(* Logix 5000 project; controller RG_Chopper vendor 1 type 14 code 235 rev 32.12; software revision 32.04 *)

TASK FLASH_1_SEC (periodic, rate 1000 ms, priority 10, watchdog 1000 ms) : FLASH
TASK MainTask (continuous, watchdog 500 ms) : MainProgram
TASK SafetyTask (periodic, rate 20 ms, priority 5, watchdog 20 ms) : SafetyProgram

MODULES
   Local : vendor 1 type 14 code 235 (5069 0, rev 32.12)
      DBX102_VFD : PowerFlex 525-EENET (Ethernet 10.0.7.41, rev 5.2, Output RPI 20 ms)   // Product Discharge Pump
      DBX104_VFD : PowerFlex 525-EENET (Ethernet 10.0.7.42, rev 5.2, Output RPI 20 ms)   // VFD DBX - 104 - Elevator Drive
           DBX104_VFD:O.Stop   // DBX-104 Drum Dumper VFD Stop
           DBX104_VFD:O.Reverse   // DBX-104 Drum Dumper VFD Direction UP
           DBX104_VFD:O.ClearFaults   // DBX-104 Drum Dumper VFD Clear Faults
           DBX104_VFD:O.Start   // DBX-104 Drum Dumper VFD Start
           DBX104_VFD:O   // DBX-104 Drum Dumper VFD Direction DOWN
      DO_4 : 5069-OB16 (5069 2, rev 2.1, StandardDataDriven RPI 5 ms)   // Digital Output - Slot 4 - 16 point
           Local:2:O.Pt15.Data   // CIP Caustic Request CIP CAUSTIC CR-202
           Local:2:O.Pt14.Data   // CIP Request System Ready CIP Enable CR-201
      DI_S_3 : 5069-IB8S (5069 4, rev 1.1, SafetyInput RPI 20 ms)   // Digital Input Safety - Slot 3 - 8 point
      DI_S_4 : 5069-IB8S (5069 7, rev 1.1, SafetyInput RPI 20 ms)   // Digital Input Safety - Slot 7 - 8 point
      DI_1 : 5069-IB16 (5069 1, rev 2.1, StandardDataDriven RPI 5 ms)   // Digital Input Slot 1 - 16 point
      IO_Link_1 : vendor 322 type 12 code 1123 (Ethernet 10.0.7.71, rev 1.1, StandardDataDriven RPI 10 ms)   // I/O-Link #1 - AL1123
           IO_Link_1:I.Data[207].8   // Port 0 LS-U1
           IO_Link_1:I.Data[207].0   // Port 1 LSS-U2
           IO_Link_1:I.Data[207].10   // Port 4 LS-OT
           IO_Link_1:I.Data[207].1   // Port 3 LS-L1
           IO_Link_1:I.Data[207].9   // Port 2 LSS-L2
      DI_S_2 : 5069-IB8S (5069 3, rev 1.1, SafetyInput RPI 20 ms)   // Digital Input Safety - Slot 2 - 8 point
      DO_S_5 : 5069-OBV8S (5069 5, rev 1.11, SafetyOutput RPI 20 ms, SafetyInput RPI 20 ms)   // Digital Output Safety - Slot 5 - 8 point
           Local:5:O.Pt05.Data   // M104 Elevator Motor Start FORWARD UP (Safety)
           Local:5:O.Pt02.Data   // Reset Button Light
           Local:5:O.Pt03.Data   // Interface Relay Output
           Local:5:O.Pt06.Data   // M104 Elevator Motor Start REVERSE (Safety)
           Local:5:O.Pt04.Data   // M104 Elevator Motor Start (EN) (Safety)
      AO_6 : vendor 1 type 115 code 313 (5069 6, rev 2.1, StandardDataDriven RPI 80 ms)   // Analog Output - Slot 6 - 8 point
END_MODULES

ADD_ON_INSTRUCTION ANLG_SCALE   (* revision 1.0, vendor JBT Food Tech *)
// Scales an Analog Value
// Revision note:
// Rev 1.0 - 9/9/2010 - KM
VAR_INPUT
   Anlg_In : REAL; {required}
   RAW_Min : REAL; {visible}
   RAW_Max : REAL; {visible}
   EU_Min : REAL; {visible}
   EU_Max : REAL; {visible}
END_VAR
VAR_OUTPUT
   Anlg_Scaled : REAL; {access Read Only, required}
END_VAR

ROUTINE Logic   (* ladder *)
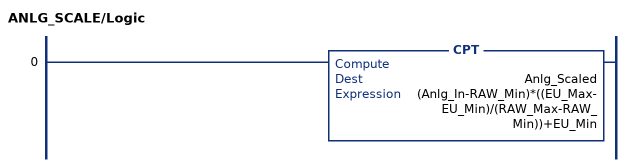
   0: CPT(Anlg_Scaled,(Anlg_In-RAW_Min)*((EU_Max-EU_Min)/(RAW_Max-RAW_Min))+EU_Min);
END_ROUTINE
END_ADD_ON_INSTRUCTION

ADD_ON_INSTRUCTION Generic_4PORT_IOL   (* revision 1.0 *)
// Revision note:
// 4/27/17
VAR_OUTPUT
   Datastorage_Error : BOOL; {access Read Only, visible}
   Device_Not_Connected : BOOL; {access Read Only, visible}
   Invalid_Data : BOOL; {access Read Only, visible}
   IOL_Mode : BOOL; {access Read Only, visible}
END_VAR
VAR_IN_OUT
   PLC_Input : INT[123]; {required}
   PLC_Output : INT[87]; {required}
END_VAR
VAR_INPUT
   Port_Process_Data_Size : INT; {visible}
   Port_Number : INT; {visible}
END_VAR
VAR_OUTPUT
   Process_Data : INT; {access Read Only}
   Wrong_VID_DID : BOOL; {access Read Only, visible}
   IN_Data1 : INT; {visible}
   IN_Data2 : INT; {visible}
   IN_Data3 : INT; {visible}
   IN_Data4 : INT; {visible}
   Out_Data1 : INT; {visible}
   Out_Data2 : INT; {visible}
   Out_Data3 : INT; {visible}
   Out_Data4 : INT; {visible}
   Vendor_ID : INT; {access Read Only, visible}
   Device_ID : INT; {access Read Only, visible}
END_VAR
VAR
   Data_Size : INT; {access None}
   Offset_Address : INT; {access None}
   Offset_StatusFlgs : INT; {access None}
   Process_Offset : INT; {access None}
   Process_PDI : INT; {access None}
   RealPort_Num : INT; {access None}
   StatusFlgs_Offset : INT; {access None}
   Process_Out_Offset : INT; {access None}
END_VAR

ROUTINE Logic   (* ladder *)
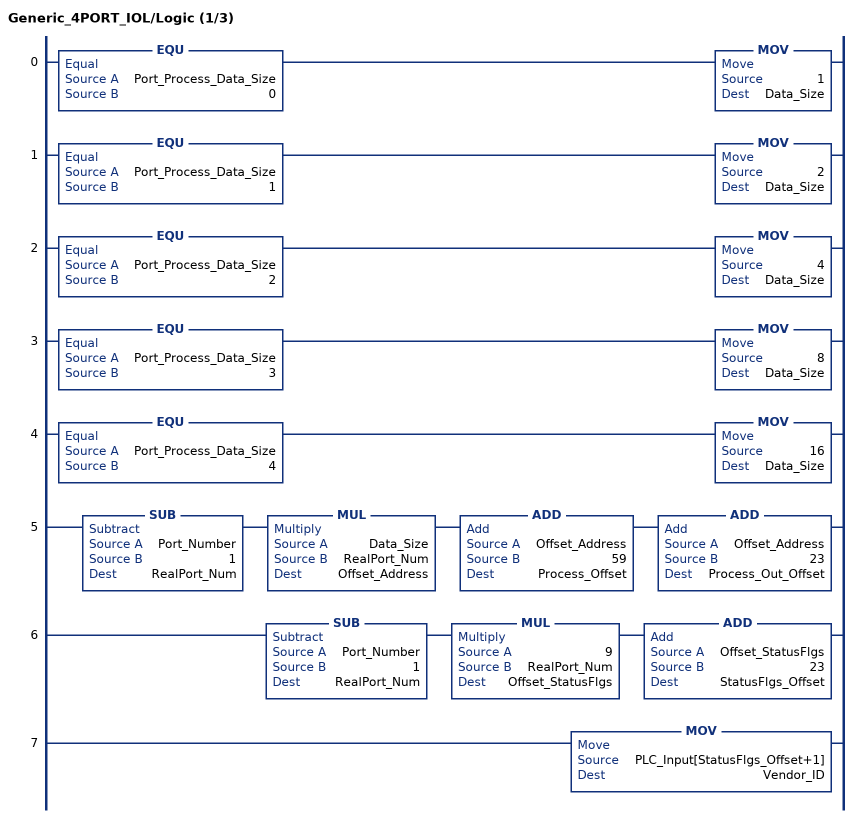
   0: EQU(Port_Process_Data_Size,0)MOV(1,Data_Size);
   1: EQU(Port_Process_Data_Size,1)MOV(2,Data_Size);
   2: EQU(Port_Process_Data_Size,2)MOV(4,Data_Size);
   3: EQU(Port_Process_Data_Size,3)MOV(8,Data_Size);
   4: EQU(Port_Process_Data_Size,4)MOV(16,Data_Size);
   5: SUB(Port_Number,1,RealPort_Num)MUL(Data_Size,RealPort_Num,Offset_Address)ADD(Offset_Address,59,Process_Offset)ADD(Offset_Address,23,Process_Out_Offset);
   6: SUB(Port_Number,1,RealPort_Num)MUL(9,RealPort_Num,Offset_StatusFlgs)ADD(Offset_StatusFlgs,23,StatusFlgs_Offset);
   7: MOV(PLC_Input[StatusFlgs_Offset+1],Vendor_ID);
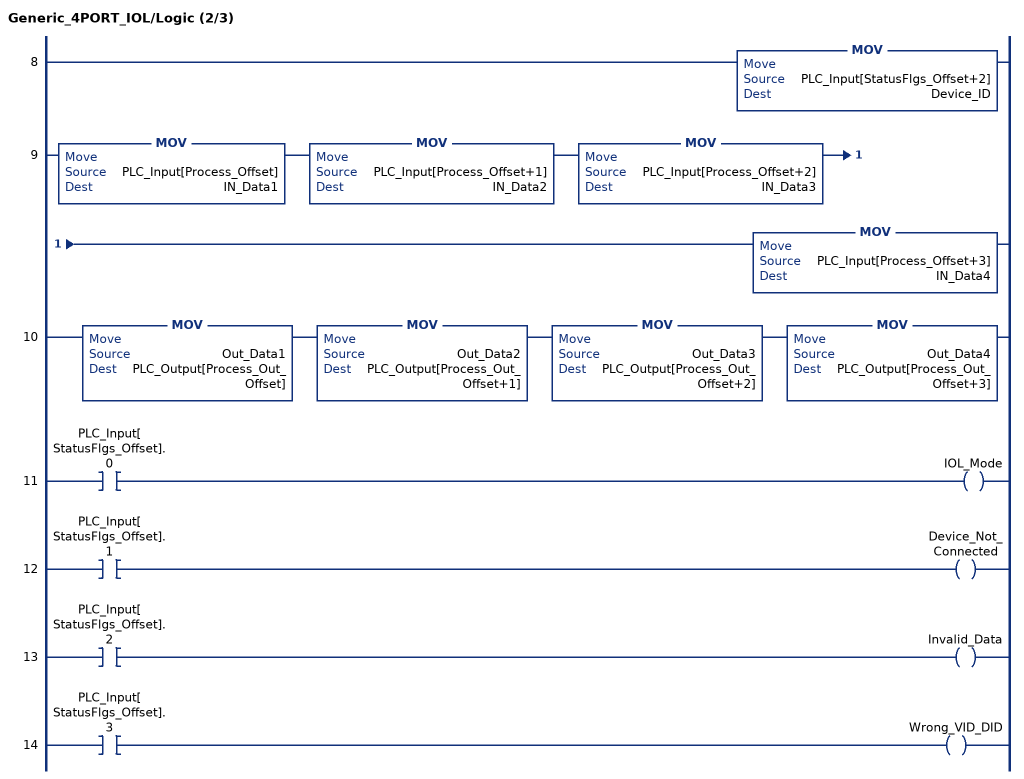
   8: MOV(PLC_Input[StatusFlgs_Offset+2],Device_ID);
   9: MOV(PLC_Input[Process_Offset],IN_Data1)MOV(PLC_Input[Process_Offset+1],IN_Data2)MOV(PLC_Input[Process_Offset+2],IN_Data3)MOV(PLC_Input[Process_Offset+3],IN_Data4);
   10: MOV(Out_Data1,PLC_Output[Process_Out_Offset])MOV(Out_Data2,PLC_Output[Process_Out_Offset+1])MOV(Out_Data3,PLC_Output[Process_Out_Offset+2])MOV(Out_Data4,PLC_Output[Process_Out_Offset+3]);
   11: XIC(PLC_Input[StatusFlgs_Offset].0)OTE(IOL_Mode);
   12: XIC(PLC_Input[StatusFlgs_Offset].1)OTE(Device_Not_Connected);
   13: XIC(PLC_Input[StatusFlgs_Offset].2)OTE(Invalid_Data);
   14: XIC(PLC_Input[StatusFlgs_Offset].3)OTE(Wrong_VID_DID);
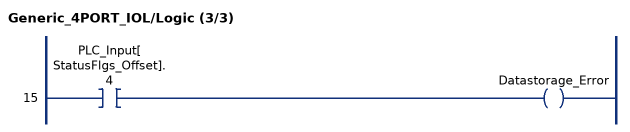
   15: XIC(PLC_Input[StatusFlgs_Offset].4)OTE(Datastorage_Error);
END_ROUTINE
END_ADD_ON_INSTRUCTION

ADD_ON_INSTRUCTION Generic_8PORT_IOL   (* revision 1.0 *)
// Revision note:
// 4/27/17
VAR_OUTPUT
   Datastorage_Error : BOOL; {access Read Only, visible}
   Device_Not_Connected : BOOL; {access Read Only, visible}
   Invalid_Data : BOOL; {access Read Only, visible}
   IOL_Mode : BOOL; {access Read Only, visible}
END_VAR
VAR_IN_OUT
   PLC_Input : INT[223]; {required}
   PLC_Output : INT[151]; {required}
END_VAR
VAR_INPUT
   Port_Process_Data_Size : INT; {visible}
   Port_Number : INT; {visible}
END_VAR
VAR_OUTPUT
   Process_Data : INT; {access Read Only}
   Wrong_VID_DID : BOOL; {access Read Only, visible}
   IN_Data1 : INT; {visible}
   IN_Data2 : INT; {visible}
   IN_Data3 : INT; {visible}
   IN_Data4 : INT; {visible}
   Out_Data1 : INT; {visible}
   Out_Data2 : INT; {visible}
   Out_Data3 : INT; {visible}
   Out_Data4 : INT; {visible}
   Vendor_ID : INT; {access Read Only, visible}
   Device_ID : INT; {access Read Only, visible}
END_VAR
VAR
   Data_Size : INT; {access None}
   Offset_Address : INT; {access None}
   Offset_StatusFlgs : INT; {access None}
   Process_Offset : INT; {access None}
   Process_PDI : INT; {access None}
   RealPort_Num : INT; {access None}
   StatusFlgs_Offset : INT; {access None}
   Process_Out_Offset : INT; {access None}
END_VAR

ROUTINE Logic   (* ladder *)
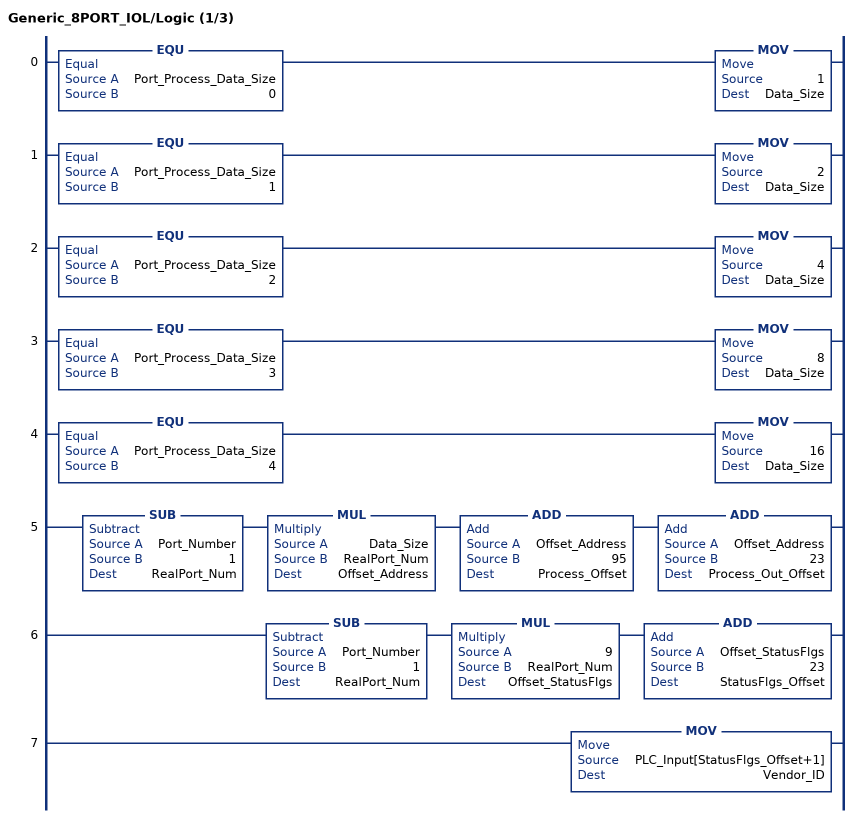
   0: EQU(Port_Process_Data_Size,0)MOV(1,Data_Size);
   1: EQU(Port_Process_Data_Size,1)MOV(2,Data_Size);
   2: EQU(Port_Process_Data_Size,2)MOV(4,Data_Size);
   3: EQU(Port_Process_Data_Size,3)MOV(8,Data_Size);
   4: EQU(Port_Process_Data_Size,4)MOV(16,Data_Size);
   5: SUB(Port_Number,1,RealPort_Num)MUL(Data_Size,RealPort_Num,Offset_Address)ADD(Offset_Address,95,Process_Offset)ADD(Offset_Address,23,Process_Out_Offset);
   6: SUB(Port_Number,1,RealPort_Num)MUL(9,RealPort_Num,Offset_StatusFlgs)ADD(Offset_StatusFlgs,23,StatusFlgs_Offset);
   7: MOV(PLC_Input[StatusFlgs_Offset+1],Vendor_ID);
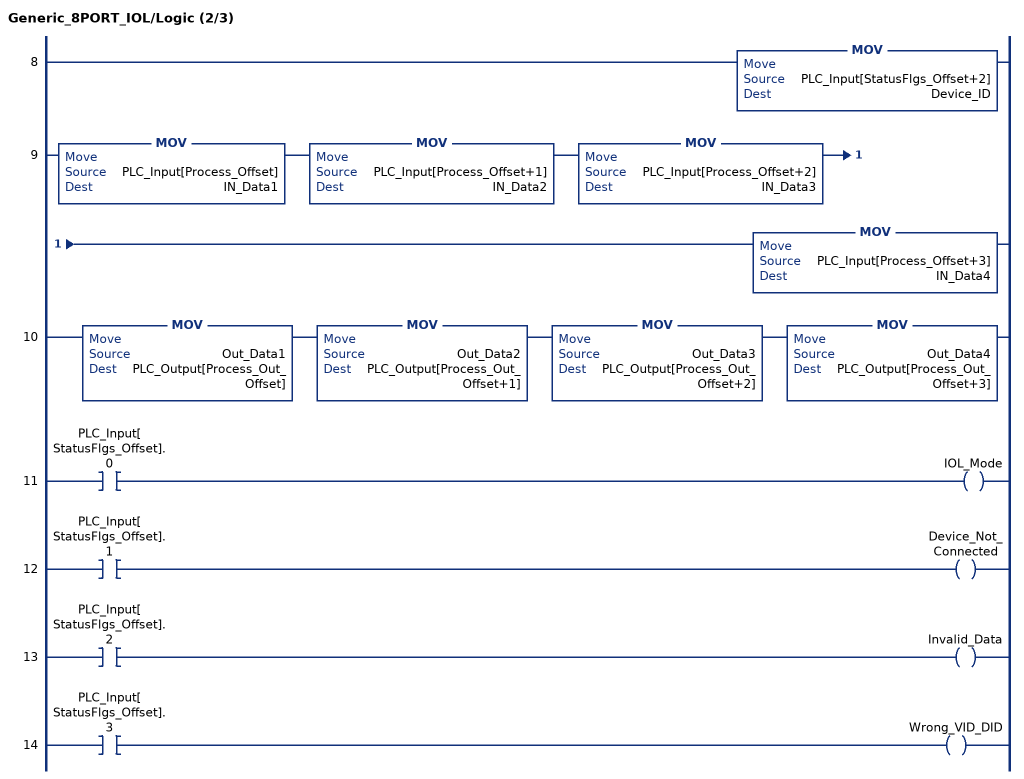
   8: MOV(PLC_Input[StatusFlgs_Offset+2],Device_ID);
   9: MOV(PLC_Input[Process_Offset],IN_Data1)MOV(PLC_Input[Process_Offset+1],IN_Data2)MOV(PLC_Input[Process_Offset+2],IN_Data3)MOV(PLC_Input[Process_Offset+3],IN_Data4);
   10: MOV(Out_Data1,PLC_Output[Process_Out_Offset])MOV(Out_Data2,PLC_Output[Process_Out_Offset+1])MOV(Out_Data3,PLC_Output[Process_Out_Offset+2])MOV(Out_Data4,PLC_Output[Process_Out_Offset+3]);
   11: XIC(PLC_Input[StatusFlgs_Offset].0)OTE(IOL_Mode);
   12: XIC(PLC_Input[StatusFlgs_Offset].1)OTE(Device_Not_Connected);
   13: XIC(PLC_Input[StatusFlgs_Offset].2)OTE(Invalid_Data);
   14: XIC(PLC_Input[StatusFlgs_Offset].3)OTE(Wrong_VID_DID);
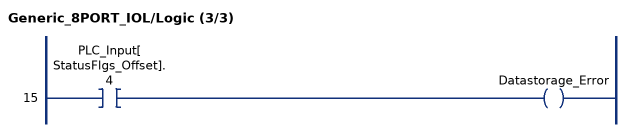
   15: XIC(PLC_Input[StatusFlgs_Offset].4)OTE(Datastorage_Error);
END_ROUTINE
END_ADD_ON_INSTRUCTION

ADD_ON_INSTRUCTION HOA_CTRL   (* revision 1.0, vendor JBT Food Tech *)
// Device Control - Hand, Off, Auto
// Revision note:
// Rev 1.0 - 9/7/2010 - KM
VAR_INPUT
   AUTO_ALL : BOOL; {required}   // Global Device Auto
   Auto_PB : BOOL;   // - Auto Push Button
   Man_PB : BOOL;   // - Manual Push Button
   Off_PB : BOOL;   // - Off Push Button
END_VAR
VAR_OUTPUT
   Auto : BOOL; {visible}   // - Auto Mode
   Man : BOOL; {visible}   // - Manual Mode
   Off : BOOL; {visible}   // - Off Mode
END_VAR
VAR_INPUT
   Dev_DIS : BOOL; {required}   // Device Disable (E-Stop?)
   Auto_Run : BOOL; {visible}   // - Auto Mode Output Control
END_VAR
VAR_OUTPUT
   Output : BOOL; {access Read Only, required}   // - Device Output
END_VAR
VAR_INPUT
   FB_EN : BOOL; {visible}   // Feed Back Fault Enabled
END_VAR
VAR_OUTPUT
   Fault_AL : BOOL; {required}   // Device Fault Alarm
END_VAR
VAR_INPUT
   Fault_INH : BOOL; {visible}   // Device Fault Alarm Inhibit
   Aux_FB : BOOL; {required}   // - Device AUXillary Feed Back
   Fault_ACK : BOOL; {required}   // Device Fault Acknowlege
   Man_INH : BOOL; {access None, visible}   // - Manual Function Inhibit
   STOP : BOOL; {access None, required}   // - Global Stop
END_VAR
VAR
   Flt_Tmr : TIMER := (PRE := 10000); {access None}   // Fault Timer
END_VAR

ROUTINE Logic   (* ladder *)
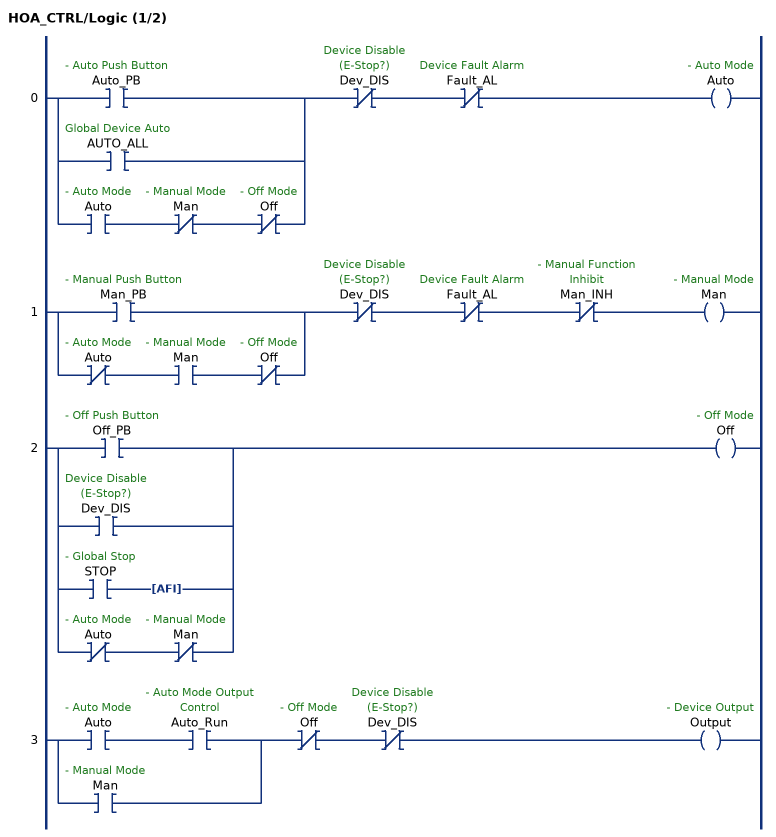
   0: [XIC(Auto_PB) ,XIC(AUTO_ALL) ,XIC(Auto) XIO(Man) XIO(Off) ]XIO(Dev_DIS)XIO(Fault_AL)OTE(Auto);
   1: [XIC(Man_PB) ,XIO(Auto) XIC(Man) XIO(Off) ]XIO(Dev_DIS)XIO(Fault_AL)XIO(Man_INH)OTE(Man);
   2: [XIC(Off_PB) ,XIC(Dev_DIS) ,XIC(STOP) AFI() ,XIO(Auto) XIO(Man) ]OTE(Off);
   3: [XIC(Auto) XIC(Auto_Run) ,XIC(Man) ]XIO(Off)XIO(Dev_DIS)OTE(Output);
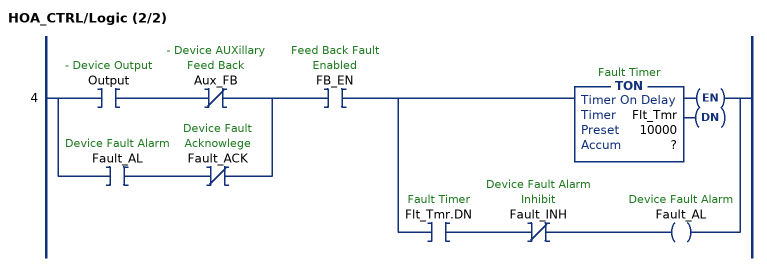
   4: [XIC(Output) XIO(Aux_FB) ,XIC(Fault_AL) XIO(Fault_ACK) ]XIC(FB_EN)[TON(Flt_Tmr,?,?) ,XIC(Flt_Tmr.DN) XIO(Fault_INH) OTE(Fault_AL) ];
END_ROUTINE
END_ADD_ON_INSTRUCTION

ADD_ON_INSTRUCTION HOA_CTRL_v2   (* revision 2.0, vendor JBT Food Tech *)
// Device Control - Hand, Off, Auto
// with Two Button Control Option
// Revision note:
// Rev 2.0 - 12/18/2017 - KM
// Help:
// When Two_Btn_EN = 1 the  two bools TB_AM and TB_MAN_Strt are enabled for use.
// Both controls require an external PUSH-PUSH ( latched toggle ) to function properly.
// The TB_AM button when OFF selects AUTO, when ON selects MANUAL.
// The TB_MAN_Strt when ON starts motor, when OFF stops motor.
// This block is backward compatible with V1.0.
VAR_INPUT
   AUTO_ALL : BOOL; {required}   // Global Device Auto
   Auto_PB : BOOL;   // - Auto Push Button
   Man_PB : BOOL;   // - Manual Push Button
   Off_PB : BOOL;   // - Off Push Button
END_VAR
VAR_OUTPUT
   Auto : BOOL; {visible}   // - Auto Mode
   Man : BOOL; {visible}   // - Manual Mode
   Off : BOOL; {visible}   // - Off Mode
END_VAR
VAR_INPUT
   Dev_DIS : BOOL; {visible}   // Device Disable (E-Stop?)
   Auto_Run : BOOL; {visible}   // - Auto Mode Output Control
END_VAR
VAR_OUTPUT
   Output : BOOL; {access Read Only, required}   // - Device Output
END_VAR
VAR_INPUT
   FB_EN : BOOL; {visible}   // Feed Back Fault Enabled
END_VAR
VAR_OUTPUT
   Fault_AL : BOOL; {access Read Only, required}   // Device Fault Alarm
END_VAR
VAR_INPUT
   Fault_INH : BOOL; {visible}   // Device Fault Alarm Inhibit
   Aux_FB : BOOL; {required}   // - Device AUXillary Feed Back
   Fault_ACK : BOOL; {required}   // Device Fault Acknowlege
   Man_INH : BOOL; {access None, visible}   // - Manual Function Inhibit
   STOP : BOOL; {access None, required}   // - Global Stop
   Two_Btn_EN : BOOL; {visible}   // Two Button Control Enabled
   TB_AM : BOOL; {required}   // Two Button Control Auto / Man (Requires Push-Push) ( Auto = 0 )
   TB_MAN_Srt : BOOL; {required}   // Two Button Control Manal Start Latch (1= Start, 2= Stop) (Requires Push-Push)
END_VAR
VAR
   Flt_Tmr : TIMER := (PRE := 10000); {access None}   // Fault Timer
   ONS : DINT; {access None}   // One Shot Word
END_VAR

ROUTINE Logic   (* ladder *)
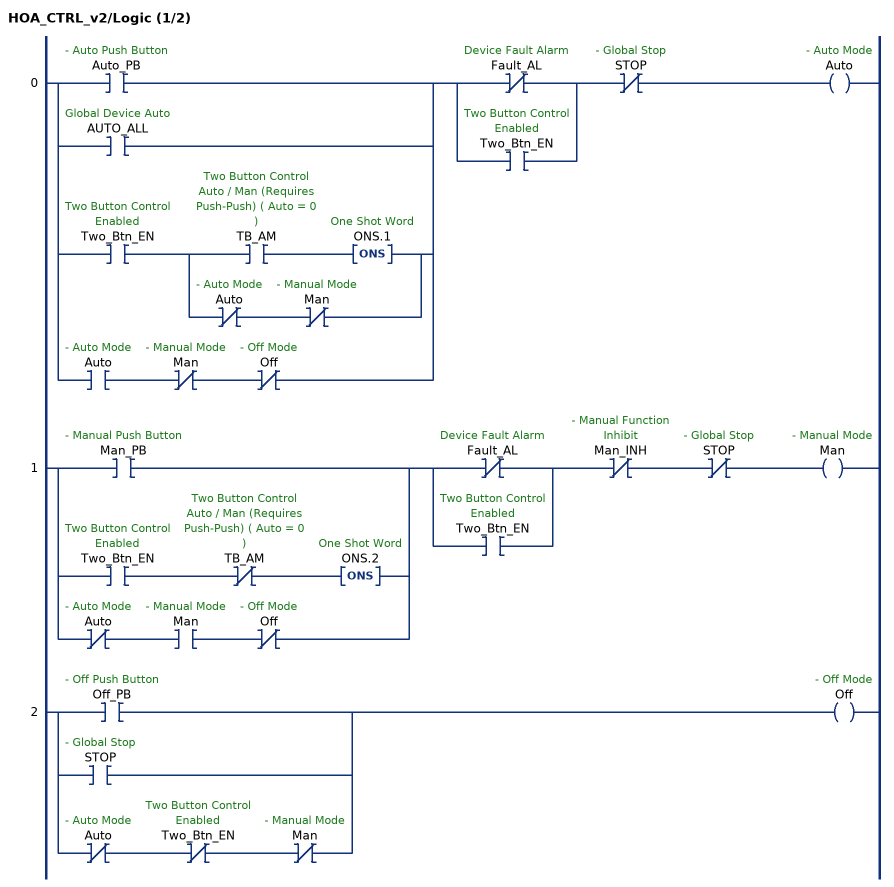
   0: [XIC(Auto_PB) ,XIC(AUTO_ALL) ,XIC(Two_Btn_EN) [XIC(TB_AM) ONS(ONS.1) ,XIO(Auto) XIO(Man) ] ,XIC(Auto) XIO(Man) XIO(Off) ][XIO(Fault_AL) ,XIC(Two_Btn_EN) ]XIO(STOP)OTE(Auto);
   1: [XIC(Man_PB) ,XIC(Two_Btn_EN) XIO(TB_AM) ONS(ONS.2) ,XIO(Auto) XIC(Man) XIO(Off) ][XIO(Fault_AL) ,XIC(Two_Btn_EN) ]XIO(Man_INH)XIO(STOP)OTE(Man);
   2: [XIC(Off_PB) ,XIC(STOP) ,XIO(Auto) XIO(Two_Btn_EN) XIO(Man) ]OTE(Off);
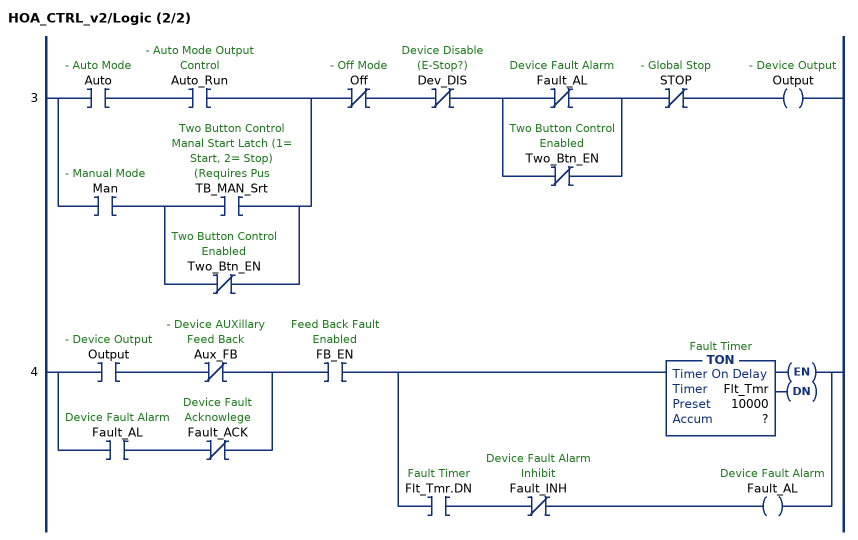
   3: [XIC(Auto) XIC(Auto_Run) ,XIC(Man) [XIC(TB_MAN_Srt) ,XIO(Two_Btn_EN) ] ]XIO(Off)XIO(Dev_DIS)[XIO(Fault_AL) ,XIO(Two_Btn_EN) ]XIO(STOP)OTE(Output);
   4: [XIC(Output) XIO(Aux_FB) ,XIC(Fault_AL) XIO(Fault_ACK) ]XIC(FB_EN)[TON(Flt_Tmr,?,?) ,XIC(Flt_Tmr.DN) XIO(Fault_INH) OTE(Fault_AL) ];
END_ROUTINE
END_ADD_ON_INSTRUCTION

ADD_ON_INSTRUCTION PN_PI_PP_4PORT_IOL   (* revision 1.0, vendor ifm efector *)
// Cyclic Data with Diagnostics
// Revision note:
// 4/27/17
VAR_IN_OUT
   PLC_Input : INT[123]; {required}
END_VAR
VAR_INPUT
   Port_Process_Data_Size : INT := 4; {visible}
   Port_Number : INT; {visible}
END_VAR
VAR_OUTPUT
   Datastorage_Error : BOOL; {access Read Only, visible}
   Process_Data : INT; {access Read Only}
   Device_Not_Connected : BOOL; {access Read Only, visible}
   IOL_Mode : BOOL; {access Read Only, visible}
   Invalid_Data : BOOL; {access Read Only, visible}
   Wrong_VID_DID : BOOL; {access Read Only, visible}
   Out1 : BOOL; {access Read Only, visible}
END_VAR
VAR_INPUT
   Pressure_Gradient : REAL := 0.1; {visible}
END_VAR
VAR_OUTPUT
   Pressure : REAL; {visible}
   Vendor_ID : INT; {access Read Only, visible}
   Device_ID : INT; {access Read Only, visible}
   Out2 : BOOL; {access Read Only, visible}
END_VAR
VAR
   RealPort_Num : INT; {access None}
   Offset_Address : INT; {access None}
   Process_PDI : INT; {access None}
   Process_Offset : INT; {access None}
   Offset_StatusFlgs : INT; {access None}
   StatusFlgs_Offset : INT; {access None}
   Data_Size : INT; {access None}
   Pressure_msk : INT; {access None}
END_VAR

ROUTINE Logic   (* ladder *)
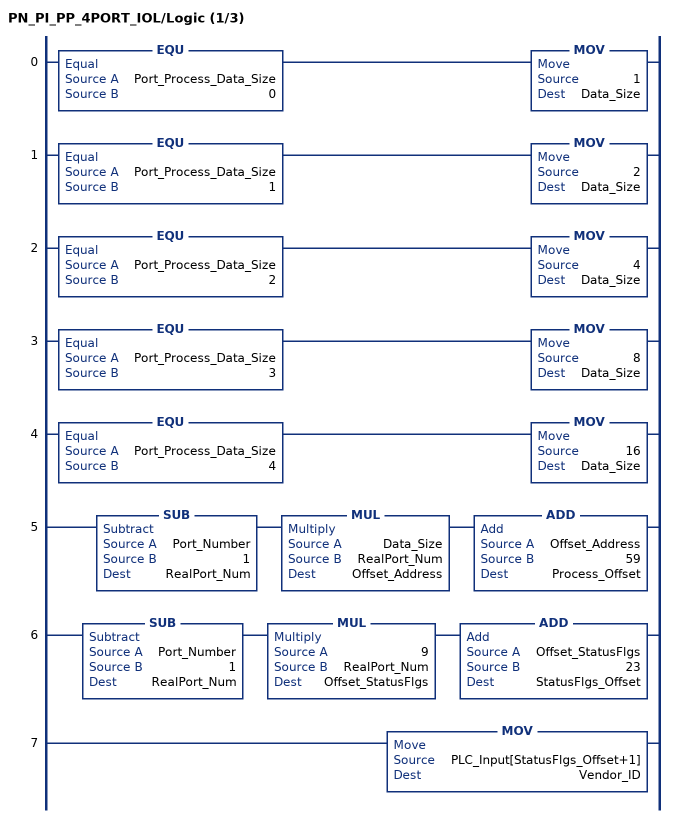
   0: EQU(Port_Process_Data_Size,0)MOV(1,Data_Size);
   1: EQU(Port_Process_Data_Size,1)MOV(2,Data_Size);
   2: EQU(Port_Process_Data_Size,2)MOV(4,Data_Size);
   3: EQU(Port_Process_Data_Size,3)MOV(8,Data_Size);
   4: EQU(Port_Process_Data_Size,4)MOV(16,Data_Size);
   5: SUB(Port_Number,1,RealPort_Num)MUL(Data_Size,RealPort_Num,Offset_Address)ADD(Offset_Address,59,Process_Offset);
   6: SUB(Port_Number,1,RealPort_Num)MUL(9,RealPort_Num,Offset_StatusFlgs)ADD(Offset_StatusFlgs,23,StatusFlgs_Offset);
   7: MOV(PLC_Input[StatusFlgs_Offset+1],Vendor_ID);
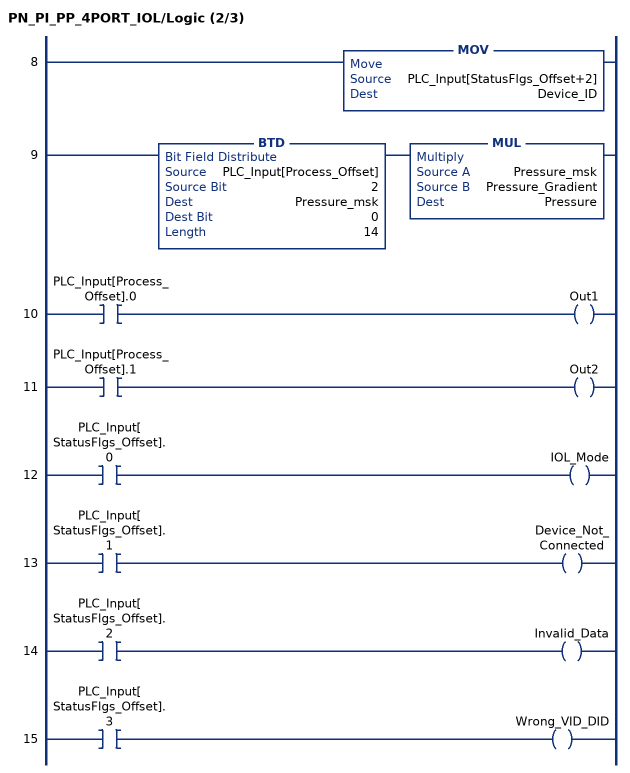
   8: MOV(PLC_Input[StatusFlgs_Offset+2],Device_ID);
   9: BTD(PLC_Input[Process_Offset],2,Pressure_msk,0,14)MUL(Pressure_msk,Pressure_Gradient,Pressure);
   10: XIC(PLC_Input[Process_Offset].0)OTE(Out1);
   11: XIC(PLC_Input[Process_Offset].1)OTE(Out2);
   12: XIC(PLC_Input[StatusFlgs_Offset].0)OTE(IOL_Mode);
   13: XIC(PLC_Input[StatusFlgs_Offset].1)OTE(Device_Not_Connected);
   14: XIC(PLC_Input[StatusFlgs_Offset].2)OTE(Invalid_Data);
   15: XIC(PLC_Input[StatusFlgs_Offset].3)OTE(Wrong_VID_DID);
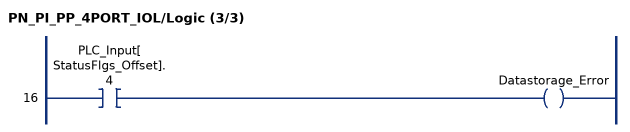
   16: XIC(PLC_Input[StatusFlgs_Offset].4)OTE(Datastorage_Error);
END_ROUTINE
END_ADD_ON_INSTRUCTION

ADD_ON_INSTRUCTION PN_PI_PP_8PORT_IOL   (* revision 1.0, vendor ifm efector *)
// Cyclic Data with Diagnostics
// Revision note:
// 4/27/17
VAR_IN_OUT
   PLC_Input : INT[223]; {required}
END_VAR
VAR_INPUT
   Port_Process_Data_Size : INT := 4; {visible}
   Port_Number : INT; {visible}
END_VAR
VAR_OUTPUT
   Datastorage_Error : BOOL; {access Read Only, visible}
   Process_Data : INT; {access Read Only}
   Device_Not_Connected : BOOL; {access Read Only, visible}
   IOL_Mode : BOOL; {access Read Only, visible}
   Invalid_Data : BOOL; {access Read Only, visible}
   Wrong_VID_DID : BOOL; {access Read Only, visible}
   Out1 : BOOL; {access Read Only, visible}
END_VAR
VAR_INPUT
   Pressure_Gradient : REAL := 0.1; {visible}
END_VAR
VAR_OUTPUT
   Pressure : REAL; {visible}
   Vendor_ID : INT; {access Read Only, visible}
   Device_ID : INT; {access Read Only, visible}
   Out2 : BOOL; {access Read Only, visible}
END_VAR
VAR
   RealPort_Num : INT; {access None}
   Offset_Address : INT; {access None}
   Process_PDI : INT; {access None}
   Process_Offset : INT; {access None}
   Offset_StatusFlgs : INT; {access None}
   StatusFlgs_Offset : INT; {access None}
   Data_Size : INT; {access None}
   Pressure_msk : INT; {access None}
END_VAR

ROUTINE Logic   (* ladder *)
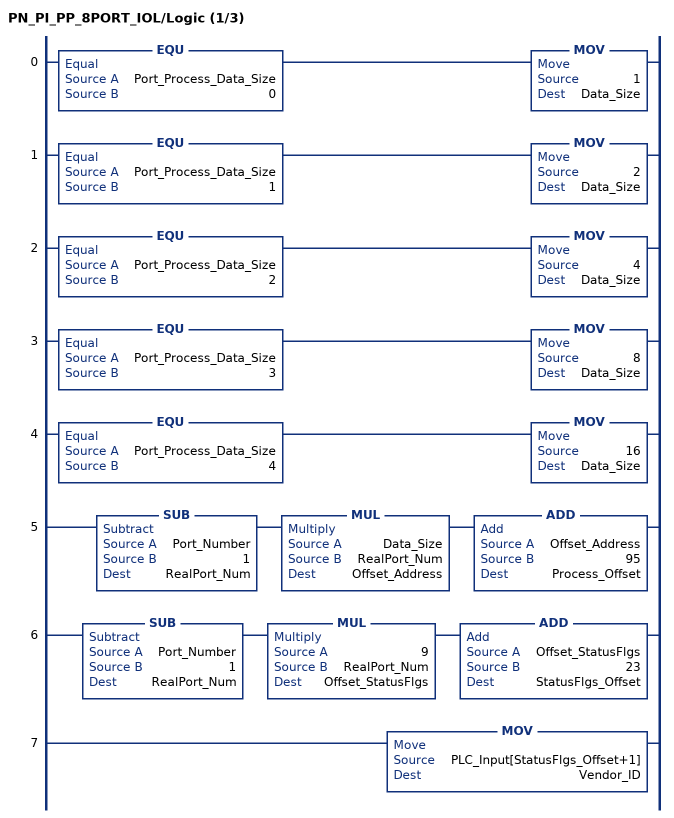
   0: EQU(Port_Process_Data_Size,0)MOV(1,Data_Size);
   1: EQU(Port_Process_Data_Size,1)MOV(2,Data_Size);
   2: EQU(Port_Process_Data_Size,2)MOV(4,Data_Size);
   3: EQU(Port_Process_Data_Size,3)MOV(8,Data_Size);
   4: EQU(Port_Process_Data_Size,4)MOV(16,Data_Size);
   5: SUB(Port_Number,1,RealPort_Num)MUL(Data_Size,RealPort_Num,Offset_Address)ADD(Offset_Address,95,Process_Offset);
   6: SUB(Port_Number,1,RealPort_Num)MUL(9,RealPort_Num,Offset_StatusFlgs)ADD(Offset_StatusFlgs,23,StatusFlgs_Offset);
   7: MOV(PLC_Input[StatusFlgs_Offset+1],Vendor_ID);
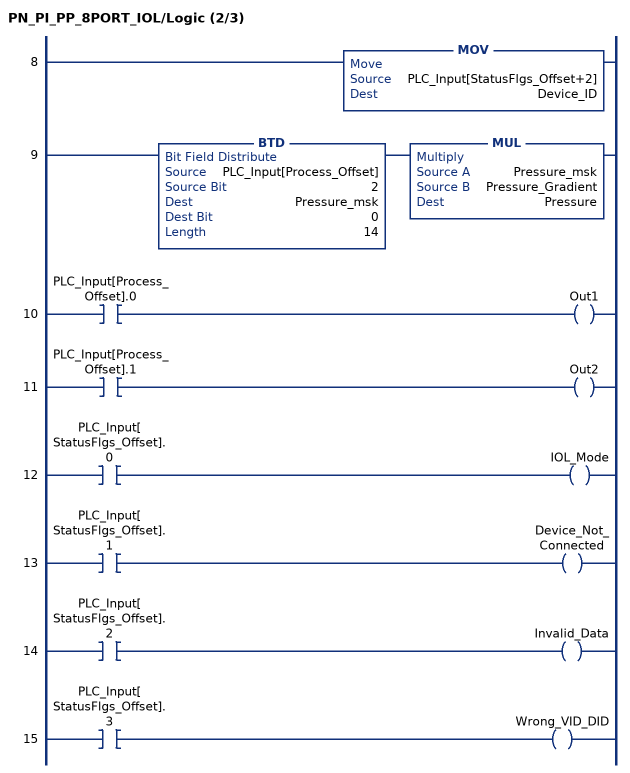
   8: MOV(PLC_Input[StatusFlgs_Offset+2],Device_ID);
   9: BTD(PLC_Input[Process_Offset],2,Pressure_msk,0,14)MUL(Pressure_msk,Pressure_Gradient,Pressure);
   10: XIC(PLC_Input[Process_Offset].0)OTE(Out1);
   11: XIC(PLC_Input[Process_Offset].1)OTE(Out2);
   12: XIC(PLC_Input[StatusFlgs_Offset].0)OTE(IOL_Mode);
   13: XIC(PLC_Input[StatusFlgs_Offset].1)OTE(Device_Not_Connected);
   14: XIC(PLC_Input[StatusFlgs_Offset].2)OTE(Invalid_Data);
   15: XIC(PLC_Input[StatusFlgs_Offset].3)OTE(Wrong_VID_DID);
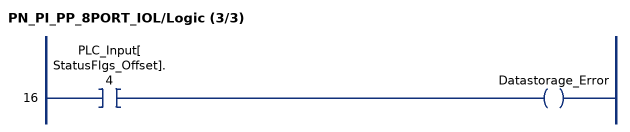
   16: XIC(PLC_Input[StatusFlgs_Offset].4)OTE(Datastorage_Error);
END_ROUTINE
END_ADD_ON_INSTRUCTION

ADD_ON_INSTRUCTION PN_PI_PP_AL1020_IOL   (* revision 1.4, vendor ifm efector *)
// Cyclic Data with Diagnostics
// Revision note:
// Supports PN2xxx, PN7xxx, PI2xxx, PPxxx
VAR_INPUT
   Port_Number : INT; {visible}
END_VAR
VAR_IN_OUT
   ioarybPLC_Input : INT[194]; {required}
END_VAR
VAR_OUTPUT
   Pressure_value : REAL; {access Read Only, required}
END_VAR
VAR_INPUT
   Pressure_value_Gradient : REAL := 0.1; {visible}
END_VAR
VAR_OUTPUT
   SwitchPoint1 : BOOL; {access Read Only, required}
   SwitchPoint2 : BOOL; {access Read Only, required}
   Vendor_ID : INT; {access Read Only, required}
   Device_ID : INT; {access Read Only, required}
   IOLinkmode_active : BOOL; {access Read Only, required}
   IOLink_communication : BOOL; {access Read Only, required}
   Device_Connected : BOOL; {access Read Only, required}
   Valid_Process_Data : BOOL; {access Read Only, required}
   Datastorage_error : BOOL; {access Read Only, required}
END_VAR
VAR
   ARYbInternInputData : INT[26]; {access None}
   Port1 : BOOL; {access None}
   Port2 : BOOL; {access None}
   Port3 : BOOL; {access None}
   Port4 : BOOL; {access None}
   Port5 : BOOL; {access None}
   Port6 : BOOL; {access None}
   Port7 : BOOL; {access None}
   Port8 : BOOL; {access None}
   Process_SWPB : INT; {access None}
   Pressure : DINT; {access None}
END_VAR

ROUTINE Logic   (* ladder *)
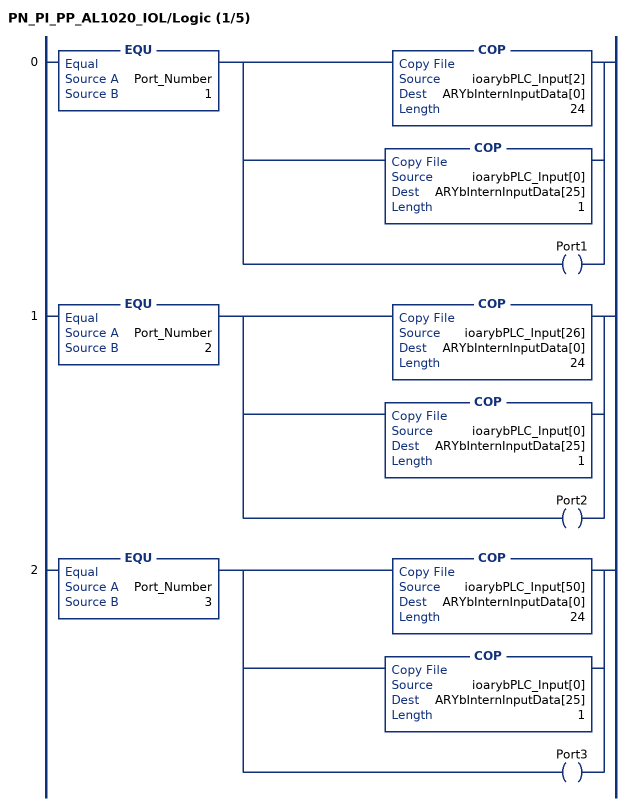
   0: EQU(Port_Number,1)[COP(ioarybPLC_Input[2],ARYbInternInputData[0],24) ,[COP(ioarybPLC_Input[0],ARYbInternInputData[25],1) ,OTE(Port1) ] ];
   1: EQU(Port_Number,2)[COP(ioarybPLC_Input[26],ARYbInternInputData[0],24) ,[COP(ioarybPLC_Input[0],ARYbInternInputData[25],1) ,OTE(Port2) ] ];
   2: EQU(Port_Number,3)[COP(ioarybPLC_Input[50],ARYbInternInputData[0],24) ,[COP(ioarybPLC_Input[0],ARYbInternInputData[25],1) ,OTE(Port3) ] ];
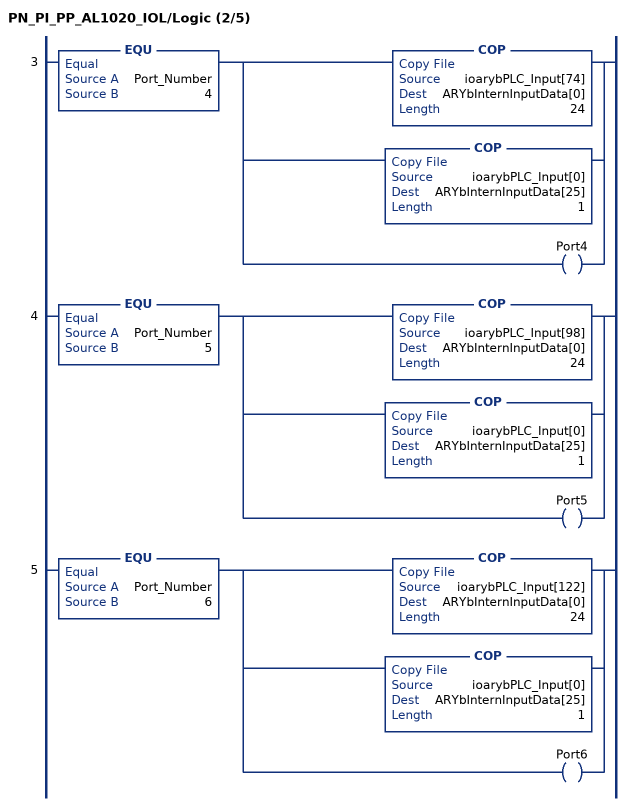
   3: EQU(Port_Number,4)[COP(ioarybPLC_Input[74],ARYbInternInputData[0],24) ,[COP(ioarybPLC_Input[0],ARYbInternInputData[25],1) ,OTE(Port4) ] ];
   4: EQU(Port_Number,5)[COP(ioarybPLC_Input[98],ARYbInternInputData[0],24) ,[COP(ioarybPLC_Input[0],ARYbInternInputData[25],1) ,OTE(Port5) ] ];
   5: EQU(Port_Number,6)[COP(ioarybPLC_Input[122],ARYbInternInputData[0],24) ,[COP(ioarybPLC_Input[0],ARYbInternInputData[25],1) ,OTE(Port6) ] ];
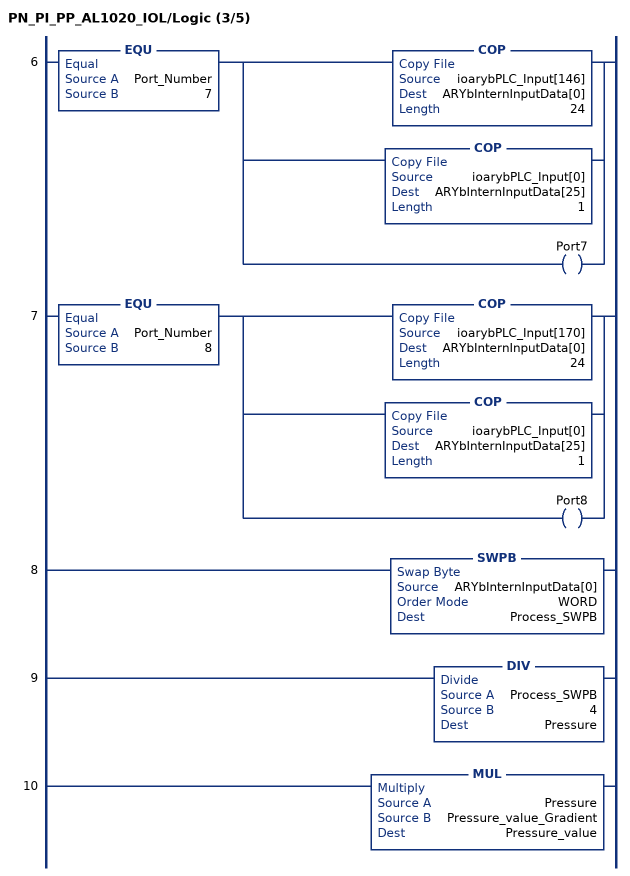
   6: EQU(Port_Number,7)[COP(ioarybPLC_Input[146],ARYbInternInputData[0],24) ,[COP(ioarybPLC_Input[0],ARYbInternInputData[25],1) ,OTE(Port7) ] ];
   7: EQU(Port_Number,8)[COP(ioarybPLC_Input[170],ARYbInternInputData[0],24) ,[COP(ioarybPLC_Input[0],ARYbInternInputData[25],1) ,OTE(Port8) ] ];
   8: SWPB(ARYbInternInputData[0],WORD,Process_SWPB);
   9: DIV(Process_SWPB,4,Pressure);
   10: MUL(Pressure,Pressure_value_Gradient,Pressure_value);
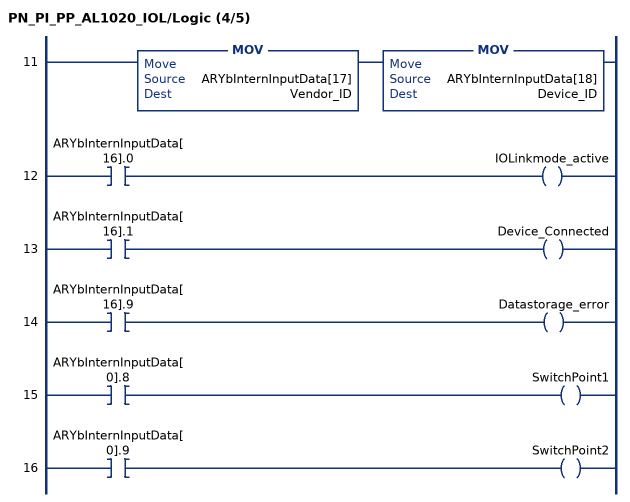
   11: MOV(ARYbInternInputData[17],Vendor_ID)MOV(ARYbInternInputData[18],Device_ID);
   12: XIC(ARYbInternInputData[16].0)OTE(IOLinkmode_active);
   13: XIC(ARYbInternInputData[16].1)OTE(Device_Connected);
   14: XIC(ARYbInternInputData[16].9)OTE(Datastorage_error);
   15: XIC(ARYbInternInputData[0].8)OTE(SwitchPoint1);
   16: XIC(ARYbInternInputData[0].9)OTE(SwitchPoint2);
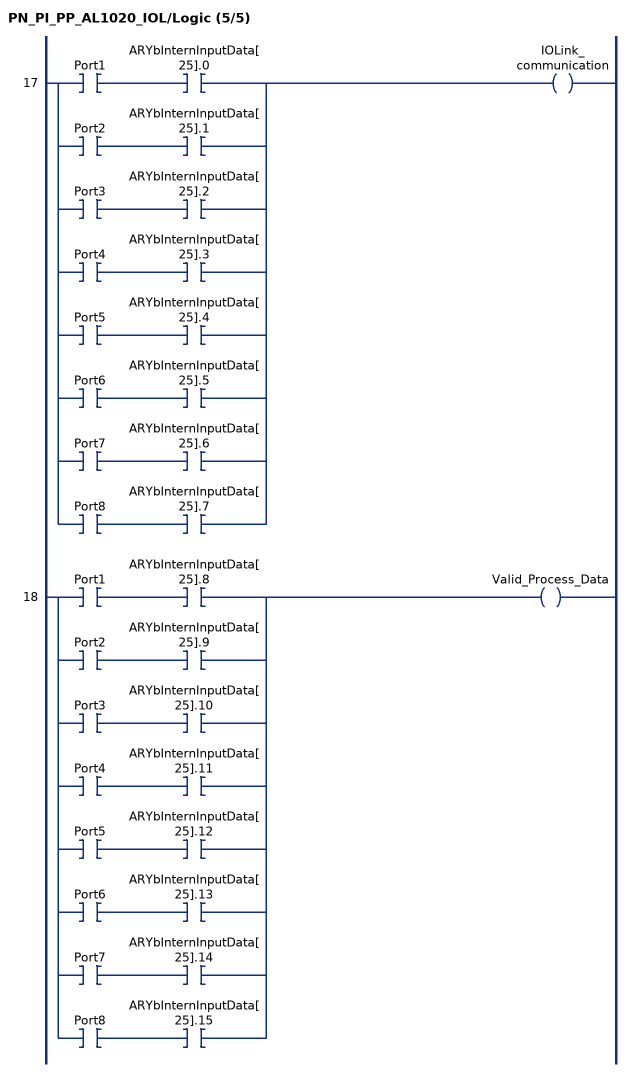
   17: [XIC(Port1) XIC(ARYbInternInputData[25].0) ,[XIC(Port2) XIC(ARYbInternInputData[25].1) ,[XIC(Port3) XIC(ARYbInternInputData[25].2) ,[XIC(Port4) XIC(ARYbInternInputData[25].3) ,[XIC(Port5) XIC(ARYbInternInputData[25].4) ,[XIC(Port6) XIC(ARYbInternInputData[25].5) ,XIC(Port7) XIC(ARYbInternInputData[25].6) ,XIC(Port8) XIC(ARYbInternInputData[25].7) ] ] ] ] ] ]OTE(IOLink_communication);
   18: [XIC(Port1) XIC(ARYbInternInputData[25].8) ,[XIC(Port2) XIC(ARYbInternInputData[25].9) ,[XIC(Port3) XIC(ARYbInternInputData[25].10) ,[XIC(Port4) XIC(ARYbInternInputData[25].11) ,[XIC(Port5) XIC(ARYbInternInputData[25].12) ,[XIC(Port6) XIC(ARYbInternInputData[25].13) ,XIC(Port7) XIC(ARYbInternInputData[25].14) ,XIC(Port8) XIC(ARYbInternInputData[25].15) ] ] ] ] ] ]OTE(Valid_Process_Data);
END_ROUTINE
END_ADD_ON_INSTRUCTION
